Universal Robots PolyScope program: shaft_insertion_back_hu_asm.urp

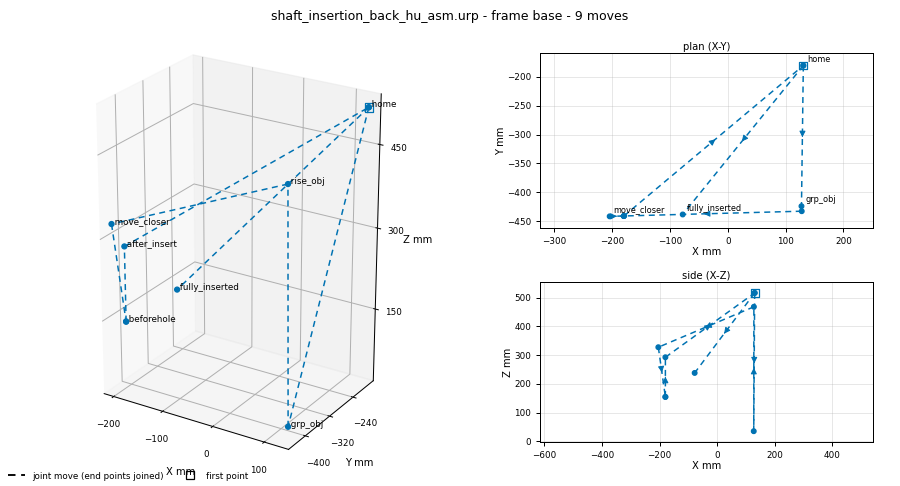
[picture p0: tool path of shaft_insertion_back_hu_asm.urp in frame base, 9 of 9 moves have a stored position in this frame; points joined in program order, loops and branches not executed]
Program shaft_insertion_back_hu_asm (installation=default directory=/programs/wrs2020 createdIn=5.7.0.90932 lastSavedIn=5.10.0.106288 robotSerialNumber=20205500607)
Calibrated DH parameters: a=[0.000096, -0.337, -0.383372, 0.000118, 0.000015, 0]; d=[0.162724, 79.377998, -95.545185, 16.300583, 0.099689, 0.099499]; alpha=[1.569249, 0.003272, 0.005201, 1.570041, -1.570219, 0]; deltaTheta=[0, 0.65664, 5.410619, 0.215927, -0.000001, 0]
Robot Program (runOnlyOnce=true)
  Folder Initialize
    MoveJ speed 180 deg/s, acceleration 80 deg/s^2 (useActiveTCP=true) feature=Base
      Waypoint home: TCP in base x=130.635 y=-180.692 z=515.97 mm, rx=-0.0117 ry=-3.1402 rz=-0.0315 rad; joints [89.951, -120.324, 80.212, -48.705, -89.957, -0.002] deg; TCP offset x=0 y=0 z=165 mm, rx=0 ry=0 rz=0 rad
    URCap Gripper (Robotiq_Grippers, Robotiq Inc.) dataModel(position=0.0, force=100.0, speed=100.0, positionInDouble=0.0, forceInDouble=100.0, speedInDouble=100.0, slaveIds=[9], blocking=true)
  MoveJ speed 60 deg/s, acceleration 80 deg/s^2 (useActiveTCP=true) feature=Base
    Waypoint grp_obj: TCP in base x=127.428 y=-423.883 z=35.422 mm, rx=-0.0117 ry=-3.1402 rz=-0.0315 rad; joints [89.401, -82.542, 128.448, -134.725, -89.783, -0.104] deg; TCP offset x=0 y=0 z=165 mm, rx=0 ry=0 rz=0 rad
  Wait Sleep waitTime=1
  URCap Gripper (Robotiq_Grippers, Robotiq Inc.) dataModel(position=100.0, force=100.0, speed=0.0, positionInDouble=100.0, forceInDouble=100.0, speedInDouble=0.0, slaveIds=[9], blocking=true)
  Wait Sleep waitTime=1
  MoveJ speed 60 deg/s, acceleration 80 deg/s^2 (useActiveTCP=true) feature=Base
    Waypoint rise_obj: TCP in base x=127.884 y=-432.566 z=467.802 mm, rx=-0.0116 ry=-3.1402 rz=-0.0314 rad; joints [89.568, -93.648, 71.545, -66.717, -89.819, -0.294] deg; TCP offset x=0 y=0 z=165 mm, rx=0 ry=0 rz=0 rad
    Waypoint move_closer: TCP in base x=-204.19 y=-441.466 z=327.291 mm, rx=-2.2399 ry=2.1904 rz=-0.0326 rad; joints [48.798, -93.225, 92.374, -88.689, -88.477, -132.668] deg; TCP offset x=0 y=0 z=165 mm, rx=0 ry=0 rz=0 rad
  MoveJ speed 60 deg/s, acceleration 80 deg/s^2 (useActiveTCP=true) feature=Base
    Waypoint beforehole: TCP in base x=-179.691 y=-440.956 z=154.622 mm, rx=2.2253 ry=-2.1669 rz=-0.0158 rad; joints [52.214, -90.414, 116.365, -117.875, -90.489, -129.348] deg; TCP offset x=0 y=0 z=165 mm, rx=0 ry=0 rz=0 rad
  MoveL speed 20 mm/s, acceleration 500 mm/s^2 (useActiveTCP=true) feature=Base
    SuppressedNode
      Waypoint athole: TCP in base x=-142.448 y=-440.96 z=154.635 mm, rx=2.2252 ry=-2.1669 rz=-0.0157 rad; joints [56.121, -92.17, 118.057, -117.755, -90.625, -125.444] deg
    MoveDirectionNode (selectedDirection=YMinus) feature=Joint_6_name
      Until TOOL_CONTACT_DETECTION (allowActions=false retraction=0 decelerationAcceleration=3 decelerationAngularAcceleration=34.906585)
  Force Frame feature=Joint_6_name; selection=[0, 1, 0, 0, 0, 0]; wrench=[0, -5, 0, 0, 0, 0]; limitsForce=[0.005, 0.01, 0.005, 1.047198, 1.047198, 1.047198]; limitsMotion=[0.1, 0.1, 0.1, 0.349066, 0.349066, 0.349066]
    Wait Sleep waitTime=3
    SuppressedNode
      Loop Counting (count=10) loopVariable(name=Loop_2)
        Force Frame feature=Base; selection=[1, 0, 1, 0, 0, 0]; wrench=[-10, 5, 5, 0, 0, 0]; limitsForce=[0.01, 0.01, 0.01, 1.047198, 1.047198, 1.047198]; limitsMotion=[0.1, 0.1, 0.1, 0.349066, 0.349066, 0.349066]
          Wait Sleep waitTime=2
        Force Frame feature=Base; selection=[1, 0, 1, 0, 0, 0]; wrench=[-10, 5, -5, 0, 0, 0]; limitsForce=[0.01, 0.01, 0.01, 1.047198, 1.047198, 1.047198]; limitsMotion=[0.1, 0.1, 0.1, 0.349066, 0.349066, 0.349066]
          Wait Sleep waitTime=2
        Force Frame feature=Base; selection=[1, 1, 0, 0, 0, 0]; wrench=[-10, 5, 5, 0, 0, 0]; limitsForce=[0.01, 0.01, 0.01, 1.047198, 1.047198, 1.047198]; limitsMotion=[0.1, 0.1, 0.1, 0.349066, 0.349066, 0.349066]
          Wait Sleep waitTime=2
        Force Frame feature=Base; selection=[1, 1, 0, 0, 0, 0]; wrench=[-10, -5, 5, 0, 0, 0]; limitsForce=[0.01, 0.01, 0.01, 1.047198, 1.047198, 1.047198]; limitsMotion=[0.1, 0.1, 0.1, 0.349066, 0.349066, 0.349066]
          Wait Sleep waitTime=2
    'spiral motion'
    SuppressedNode
      Loop Counting (count=30) loopVariable(name=Loop_1)
        MoveL speed 250 mm/s, acceleration 1200 mm/s^2 (useActiveTCP=true) feature=Base
          MoveDirectionNode (toolParams=0.005, 0.02) expression=[sin((Loop_1-1)/6*3.141),0.0,-cos((Loop_1-1)/6*3.141)]; feature=Joint_6_name
            Until DISTANCE (allowActions=false deceleration=3 distanceNodeType=STOP) Distance=0.001; motionParameters(blendRadius=0)
    'grid motion'
    loop_1 := 1
    tcp_p := get_actual_tcp_pose()
    Popup Message (haltProgram=false inputType=Variable) variable=tcp_p
    Loop While (checkContinuously=true) expression=( tcp_p[0] < -0.140) and  (loop_1 < 6)
      MoveL speed 250 mm/s, acceleration 1200 mm/s^2 (useActiveTCP=true) feature=Base
        MoveDirectionNode (selectedDirection=XPlus toolParams=0.003, 0.005) feature=Joint_6_name
          Until DISTANCE (allowActions=false deceleration=3 distanceNodeType=STOP) Distance=0.001; motionParameters(blendRadius=0)
        tcp_p := get_actual_tcp_pose()
        MoveDirectionNode (selectedDirection=ZMinus toolParams=0.003, 0.005) feature=Joint_6_name
          Until DISTANCE (allowActions=false deceleration=3 distanceNodeType=STOP) Distance=0.001; motionParameters(blendRadius=0)
        MoveDirectionNode (selectedDirection=XMinus toolParams=0.003, 0.005) feature=Joint_6_name
          Until DISTANCE (allowActions=false deceleration=3 distanceNodeType=STOP) Distance=0.001; motionParameters(blendRadius=0)
        MoveDirectionNode (selectedDirection=XMinus toolParams=0.003, 0.005) feature=Joint_6_name
          Until DISTANCE (allowActions=false deceleration=3 distanceNodeType=STOP) Distance=0.001; motionParameters(blendRadius=0)
        tcp_p := get_actual_tcp_pose()
        MoveDirectionNode (selectedDirection=ZPlus toolParams=0.003, 0.005) feature=Joint_6_name
          Until DISTANCE (allowActions=false deceleration=3 distanceNodeType=STOP) Distance=0.001; motionParameters(blendRadius=0)
        MoveDirectionNode (selectedDirection=XPlus toolParams=0.003, 0.005) feature=Joint_6_name
          Until DISTANCE (allowActions=false deceleration=3 distanceNodeType=STOP) Distance=0.001; motionParameters(blendRadius=0)
        MoveDirectionNode (selectedDirection=XPlus toolParams=0.003, 0.005) feature=Joint_6_name
          Until DISTANCE (allowActions=false deceleration=3 distanceNodeType=STOP) Distance=0.001; motionParameters(blendRadius=0)
        tcp_p := get_actual_tcp_pose()
        MoveDirectionNode (selectedDirection=ZPlus toolParams=0.003, 0.005) feature=Joint_6_name
          Until DISTANCE (allowActions=false deceleration=3 distanceNodeType=STOP) Distance=0.001; motionParameters(blendRadius=0)
        MoveDirectionNode (selectedDirection=XMinus toolParams=0.003, 0.005) feature=Joint_6_name
          Until DISTANCE (allowActions=false deceleration=3 distanceNodeType=STOP) Distance=0.001; motionParameters(blendRadius=0)
        MoveDirectionNode (selectedDirection=XMinus toolParams=0.003, 0.005) feature=Joint_6_name
          Until DISTANCE (allowActions=false deceleration=3 distanceNodeType=STOP) Distance=0.001; motionParameters(blendRadius=0)
        tcp_p := get_actual_tcp_pose()
        MoveDirectionNode (selectedDirection=ZMinus toolParams=0.003, 0.005) feature=Joint_6_name
          Until DISTANCE (allowActions=false deceleration=3 distanceNodeType=STOP) Distance=0.001; motionParameters(blendRadius=0)
        MoveDirectionNode (selectedDirection=XPlus toolParams=0.003, 0.005) feature=Joint_6_name
          Until DISTANCE (allowActions=false deceleration=3 distanceNodeType=STOP) Distance=0.001; motionParameters(blendRadius=0)
      loop_1 := loop_1+1
      tcp_p := get_actual_tcp_pose()
    Popup Message (haltProgram=false inputType=Variable) variable=tcp_p
  URCap Gripper (Robotiq_Grippers, Robotiq Inc.) dataModel(position=0.0, force=100.0, speed=100.0, positionInDouble=0.0, forceInDouble=100.0, speedInDouble=100.0, slaveIds=[9], blocking=true)
  MoveJ speed 60 deg/s, acceleration 80 deg/s^2 (useActiveTCP=true) feature=Base
    Waypoint push_shaft_rdy: TCP in base x=-179.694 y=-440.946 z=154.614 mm, rx=2.2253 ry=-2.1669 rz=-0.0157 rad; joints [52.213, -90.415, 116.367, -117.876, -90.488, -129.348] deg
  URCap Gripper (Robotiq_Grippers, Robotiq Inc.) dataModel(position=100.0, force=100.0, speed=100.0, positionInDouble=100.0, forceInDouble=100.0, speedInDouble=100.0, slaveIds=[9], blocking=true)
  SuppressedNode
    MoveL speed 10 mm/s, acceleration 1200 mm/s^2 (useActiveTCP=true) feature=Base
      Waypoint push_shaft: TCP in base x=-60.352 y=-445.424 z=219.069 mm, rx=2.1821 ry=2.2311 rz=0.0137 rad; joints [64.456, -96.881, 111.731, -104.723, -88.406, 63.074] deg
  Folder push shaft and wiggle
    Force Frame feature=Joint_6_name; selection=[0, 1, 0, 0, 0, 0]; wrench=[-20, -10, 0, 0, 0, 0]; limitsForce=[0.01, 0.01, 0.005, 1.047198, 1.047198, 1.047198]; limitsMotion=[0.1, 0.1, 0.1, 0.349066, 0.349066, 0.349066]
      Wait Sleep waitTime=1
      'grid motion'
      loop_1 := 1
      tcp_p := get_actual_tcp_pose()
      Loop While (checkContinuously=true) expression=( tcp_p[0] < -0.130) and  (loop_1 < 6)
        tcp_p := get_actual_tcp_pose()
        MoveL speed 250 mm/s, acceleration 1200 mm/s^2 (useActiveTCP=true) feature=Base
          MoveDirectionNode (selectedDirection=ZMinus toolParams=0.005, 0.02) feature=Joint_6_name
            Until DISTANCE (allowActions=false deceleration=3 distanceNodeType=STOP) Distance=0.002; motionParameters(blendRadius=0)
          tcp_p := get_actual_tcp_pose()
          MoveDirectionNode (selectedDirection=ZPlus toolParams=0.005, 0.02) feature=Joint_6_name
            Until DISTANCE (allowActions=false deceleration=3 distanceNodeType=STOP) Distance=0.002; motionParameters(blendRadius=0)
          tcp_p := get_actual_tcp_pose()
          MoveDirectionNode (selectedDirection=ZPlus toolParams=0.005, 0.02) feature=Joint_6_name
            Until DISTANCE (allowActions=false deceleration=3 distanceNodeType=STOP) Distance=0.002; motionParameters(blendRadius=0)
          tcp_p := get_actual_tcp_pose()
          MoveDirectionNode (selectedDirection=ZMinus toolParams=0.005, 0.02) feature=Joint_6_name
            Until DISTANCE (allowActions=false deceleration=3 distanceNodeType=STOP) Distance=0.002; motionParameters(blendRadius=0)
        loop_1 := loop_1+1
        tcp_p := get_actual_tcp_pose()
  MoveJ speed 60 deg/s, acceleration 80 deg/s^2 (useActiveTCP=true) feature=Base
    Waypoint after_insert: TCP in base x=-179.679 y=-440.957 z=292.449 mm, rx=2.2253 ry=-2.1669 rz=-0.0157 rad; joints [52.254, -95.603, 100.268, -96.591, -90.494, -129.429] deg
  MoveJ speed 180 deg/s, acceleration 80 deg/s^2 (useActiveTCP=true) feature=Base
    Waypoint home: TCP in base x=130.635 y=-180.692 z=515.97 mm, rx=-0.0117 ry=-3.1402 rz=-0.0315 rad; joints [89.951, -120.324, 80.212, -48.705, -89.957, -0.002] deg
  Halt
  MoveJ speed 60 deg/s, acceleration 80 deg/s^2 (useActiveTCP=true) feature=Base
    Waypoint fully_inserted: TCP in base x=-77.923 y=-438.216 z=237.961 mm, rx=2.1821 ry=2.2311 rz=0.0137 rad; joints [61.917, -98.126, 109.947, -101.635, -88.415, 60.516] deg
